(* Logix 5000 project; controller SolisPLC_Vlad_CGL1 vendor 1 type 14 code 226 rev 32.13; software revision 32.02 *)

TASK MainTask (continuous, watchdog 500 ms) : MainProgram, DataLink, Palletizer, Tutorials
TASK SafetyTask (periodic, rate 20 ms, priority 10, watchdog 20 ms, safety) : SafetyProgram

MODULES
   Local : vendor 1 type 14 code 226 (5069 0, rev 32.13)
END_MODULES

TYPE UDT_MQTT_DINT :
STRUCT
   Message : DINT;
   Delay : DINT;
   Timer : TIMER;
   RawData : DINT;
   Delta : DINT;
   OldRawData : DINT;
END_STRUCT
END_TYPE

ADD_ON_INSTRUCTION _AOI_Fah_to_Cel   (* revision 1.0 *)
VAR_INPUT
   Temperature_Fah : REAL; {required}
END_VAR
VAR_OUTPUT
   Temperature_Cel : REAL; {required}
END_VAR
VAR
   Placeholder : REAL; {access None}
   Placeholder1 : REAL; {access None}
END_VAR

ROUTINE Logic   (* ladder *)
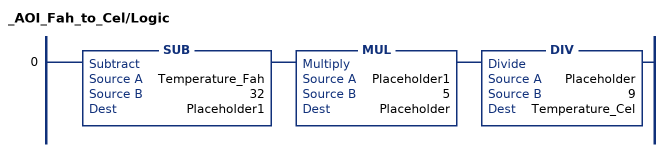
   0: SUB(Temperature_Fah,32,Placeholder1)MUL(Placeholder1,5,Placeholder)DIV(Placeholder,9,Temperature_Cel);
END_ROUTINE
END_ADD_ON_INSTRUCTION

VAR_GLOBAL   (* controller tags *)
   MQTT_OUT : UDT_MQTT_DINT[100] := ([0].Message := 2380, [0].Timer.EN := 1, [0].Timer.TT := 1, [0].RawData := 2380, [0].OldRawData := 2380, [1].Message := 10, [1].Timer.EN := 1, [1].Timer.TT := 1, [1].RawData := 10, [1].OldRawData := 10, [2].Message := 28, [2].Timer.EN := 1, [2].Timer.TT := 1, [2].RawData := 28, [2].OldRawData := 28, [3].Message := 3361, [3].Delay := 1000, [3].Timer.PRE := 1000, [3].Timer.ACC := 633, [3].Timer.EN := 1, [3].Timer.TT := 1, [3].RawData := 3994, [3].Delta := 1000, [3].OldRawData := 3361, [4].Delay := 1000, [4].Timer.PRE := 1000, [4].Timer.ACC := 994, [4].Timer.EN := 1, [4].Timer.TT := 1, [4].Delta := 1000, [5].Timer.EN := 1, [5].Timer.TT := 1, [6].Timer.EN := 1, [6].Timer.TT := 1, [7].Timer.EN := 1, [7].Timer.TT := 1, [8].Timer.EN := 1, [8].Timer.TT := 1, [9].Timer.EN := 1, [9].Timer.TT := 1, [10].Timer.EN := 1, [10].Timer.TT := 1, [11].Timer.EN := 1, [11].Timer.TT := 1, [12].Timer.EN := 1, [12].Timer.TT := 1, [13].Timer.EN := 1, [13].Timer.TT := 1, [14].Timer.EN := 1, [14].Timer.TT := 1, [15].Timer.EN := 1, [15].Timer.TT := 1, [16].Timer.EN := 1, [16].Timer.TT := 1, [17].Timer.EN := 1, [17].Timer.TT := 1, [18].Timer.EN := 1, [18].Timer.TT := 1, [19].Timer.EN := 1, [19].Timer.TT := 1,
        [20].Timer.EN := 1, [20].Timer.TT := 1, [21].Timer.EN := 1, [21].Timer.TT := 1, [22].Timer.EN := 1, [22].Timer.TT := 1, [23].Timer.EN := 1, [23].Timer.TT := 1, [24].Timer.EN := 1, [24].Timer.TT := 1, [25].Timer.EN := 1, [25].Timer.TT := 1, [26].Timer.EN := 1, [26].Timer.TT := 1, [27].Timer.EN := 1, [27].Timer.TT := 1, [28].Timer.EN := 1, [28].Timer.TT := 1, [29].Timer.EN := 1, [29].Timer.TT := 1, [30].Timer.EN := 1, [30].Timer.TT := 1, [31].Timer.EN := 1, [31].Timer.TT := 1, [32].Timer.EN := 1, [32].Timer.TT := 1, [33].Timer.EN := 1, [33].Timer.TT := 1, [34].Timer.EN := 1, [34].Timer.TT := 1, [35].Timer.EN := 1, [35].Timer.TT := 1, [36].Timer.EN := 1, [36].Timer.TT := 1, [37].Timer.EN := 1, [37].Timer.TT := 1, [38].Timer.EN := 1, [38].Timer.TT := 1, [39].Timer.EN := 1, [39].Timer.TT := 1, [40].Timer.EN := 1, [40].Timer.TT := 1, [41].Timer.EN := 1, [41].Timer.TT := 1, [42].Timer.EN := 1, [42].Timer.TT := 1, [43].Timer.EN := 1, [43].Timer.TT := 1, [44].Timer.EN := 1, [44].Timer.TT := 1, [45].Timer.EN := 1, [45].Timer.TT := 1, [46].Timer.EN := 1, [46].Timer.TT := 1, [47].Timer.EN := 1, [47].Timer.TT := 1, [48].Timer.EN := 1, [48].Timer.TT := 1, [49].Timer.EN := 1, [49].Timer.TT := 1,
        [50].Timer.EN := 1, [50].Timer.TT := 1, [51].Timer.EN := 1, [51].Timer.TT := 1, [52].Timer.EN := 1, [52].Timer.TT := 1, [53].Timer.EN := 1, [53].Timer.TT := 1, [54].Timer.EN := 1, [54].Timer.TT := 1, [55].Timer.EN := 1, [55].Timer.TT := 1, [56].Timer.EN := 1, [56].Timer.TT := 1, [57].Timer.EN := 1, [57].Timer.TT := 1, [58].Timer.EN := 1, [58].Timer.TT := 1, [59].Timer.EN := 1, [59].Timer.TT := 1, [60].Timer.EN := 1, [60].Timer.TT := 1, [61].Timer.EN := 1, [61].Timer.TT := 1, [62].Timer.EN := 1, [62].Timer.TT := 1, [63].Timer.EN := 1, [63].Timer.TT := 1, [64].Timer.EN := 1, [64].Timer.TT := 1, [65].Timer.EN := 1, [65].Timer.TT := 1, [66].Timer.EN := 1, [66].Timer.TT := 1, [67].Timer.EN := 1, [67].Timer.TT := 1, [68].Timer.EN := 1, [68].Timer.TT := 1, [69].Timer.EN := 1, [69].Timer.TT := 1, [70].Timer.EN := 1, [70].Timer.TT := 1, [71].Timer.EN := 1, [71].Timer.TT := 1, [72].Timer.EN := 1, [72].Timer.TT := 1, [73].Timer.EN := 1, [73].Timer.TT := 1, [74].Timer.EN := 1, [74].Timer.TT := 1, [75].Timer.EN := 1, [75].Timer.TT := 1, [76].Timer.EN := 1, [76].Timer.TT := 1, [77].Timer.EN := 1, [77].Timer.TT := 1, [78].Timer.EN := 1, [78].Timer.TT := 1, [79].Timer.EN := 1, [79].Timer.TT := 1,
        [80].Timer.EN := 1, [80].Timer.TT := 1, [81].Timer.EN := 1, [81].Timer.TT := 1, [82].Timer.EN := 1, [82].Timer.TT := 1, [83].Timer.EN := 1, [83].Timer.TT := 1, [84].Timer.EN := 1, [84].Timer.TT := 1, [85].Timer.EN := 1, [85].Timer.TT := 1, [86].Timer.EN := 1, [86].Timer.TT := 1, [87].Timer.EN := 1, [87].Timer.TT := 1, [88].Timer.EN := 1, [88].Timer.TT := 1, [89].Timer.EN := 1, [89].Timer.TT := 1, [90].Timer.EN := 1, [90].Timer.TT := 1, [91].Timer.EN := 1, [91].Timer.TT := 1, [92].Timer.EN := 1, [92].Timer.TT := 1, [93].Timer.EN := 1, [93].Timer.TT := 1, [94].Timer.EN := 1, [94].Timer.TT := 1, [95].Timer.EN := 1, [95].Timer.TT := 1, [96].Timer.EN := 1, [96].Timer.TT := 1, [97].Timer.EN := 1, [97].Timer.TT := 1, [98].Timer.EN := 1, [98].Timer.TT := 1, [99].Timer.EN := 1, [99].Timer.TT := 1);
   MQTT_OUT_B : DINT[100];
   MQTT_OUT_BOOL : UDT_MQTT_DINT[100] := ([0].Message := 2252, [0].RawData := 2252);
   MQTT_OUT_DINT : DINT[100] := ([0] := 30869, [1] := 30869, [2] := 10869);
   Pal_D : DINT[100] := ([0] := 2252, [1] := 10, [2] := 28);
        [0].0   // Palletizer Infeed - Start PB
        [0].1   // Palletizer Infeed - Stop PB
        [0].10   // Palletizer Discharge - Stop PB
        [0].11   // Palletizer Discharge - Running Status
        [0].12   // Palletizer Discharge - Full Pallet Ready
        [0].2   // Palletizer Infeed - Enabled Status
        [0].3   // Palletizer Infeed - Full Status
        [0].4   // Palletizer Robot - Start PB
        [0].5   // Palletizer Robot - Stop PB
        [0].6   // Palletizer Robot - Enabled Status
        [0].7   // Palletizer Robot - Pick Up Cases
        [0].8   // Palletizer Robot - Cases On Arm
        [0].9   // Palletizer Discharge - Start PB
   Pal_T : TIMER[100] := ([0].PRE := 1000, [1].PRE := 4268, [1].ACC := 4127, [1].EN := 1, [1].TT := 1, [2].PRE := 6639, [3].PRE := 7587);
   Sys_Timer : TIMER[100] := ([0].PRE := 100000, [0].ACC := 30893, [0].EN := 1, [0].TT := 1, [1].PRE := 500000, [1].ACC := 30893, [1].EN := 1, [1].TT := 1, [2].PRE := 11000, [2].ACC := 10893, [2].EN := 1, [2].TT := 1);
END_VAR

PROGRAM DataLink   (* main routine _01_Main *)
VAR
   index : DINT := 85;
END_VAR

ROUTINE _01_Main   (* ladder *)
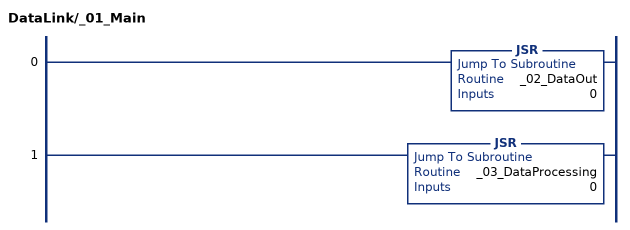
   0: JSR(_02_DataOut,0);
   1: JSR(_03_DataProcessing,0);
END_ROUTINE

ROUTINE _02_DataOut   (* ladder *)
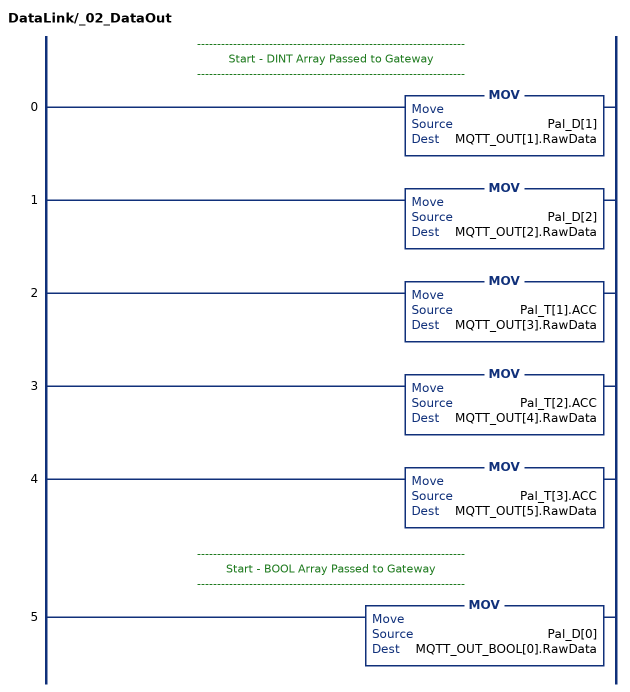
   // -------------------------------------------------------------------
   // Start - DINT Array Passed to Gateway
   // -------------------------------------------------------------------
   0: MOV(Pal_D[1],MQTT_OUT[1].RawData);
   1: MOV(Pal_D[2],MQTT_OUT[2].RawData);
   2: MOV(Pal_T[1].ACC,MQTT_OUT[3].RawData);
   3: MOV(Pal_T[2].ACC,MQTT_OUT[4].RawData);
   4: MOV(Pal_T[3].ACC,MQTT_OUT[5].RawData);
   // -------------------------------------------------------------------
   // Start - BOOL Array Passed to Gateway
   // -------------------------------------------------------------------
   5: MOV(Pal_D[0],MQTT_OUT_BOOL[0].RawData);
END_ROUTINE

ROUTINE _03_DataProcessing   (* ladder *)
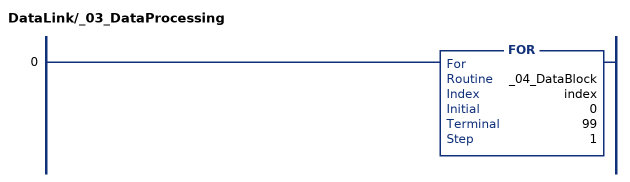
   0: FOR(_04_DataBlock,index,0,99,1);
END_ROUTINE

ROUTINE _04_DataBlock   (* ladder *)
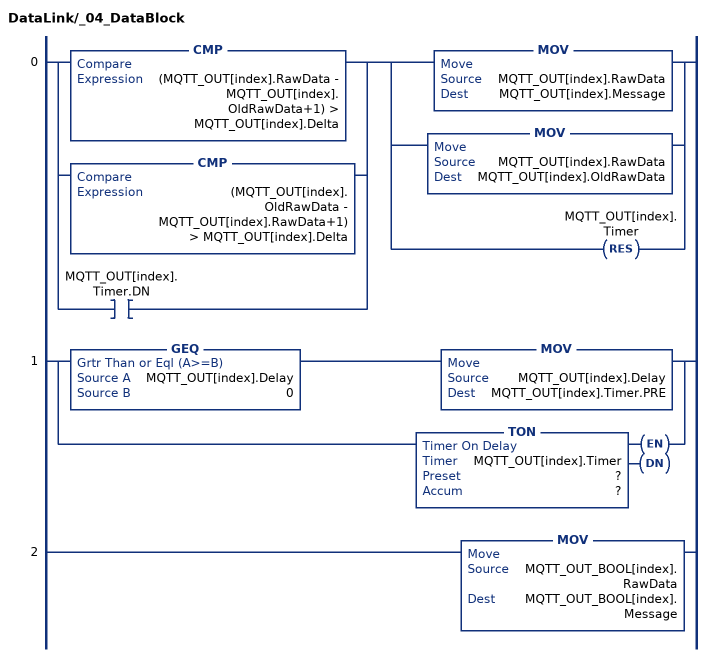
   0: [CMP((MQTT_OUT[index].RawData - MQTT_OUT[index].OldRawData+1) > MQTT_OUT[index].Delta) ,CMP((MQTT_OUT[index].OldRawData - MQTT_OUT[index].RawData+1) > MQTT_OUT[index].Delta) ,XIC(MQTT_OUT[index].Timer.DN) ][MOV(MQTT_OUT[index].RawData,MQTT_OUT[index].Message) ,MOV(MQTT_OUT[index].RawData,MQTT_OUT[index].OldRawData) ,RES(MQTT_OUT[index].Timer) ];
   1: [GEQ(MQTT_OUT[index].Delay,0) MOV(MQTT_OUT[index].Delay,MQTT_OUT[index].Timer.PRE) ,TON(MQTT_OUT[index].Timer,?,?) ];
   2: MOV(MQTT_OUT_BOOL[index].RawData,MQTT_OUT_BOOL[index].Message);
END_ROUTINE
END_PROGRAM

PROGRAM MainProgram   (* main routine MainRoutine *)

ROUTINE MainRoutine   (* ladder *)
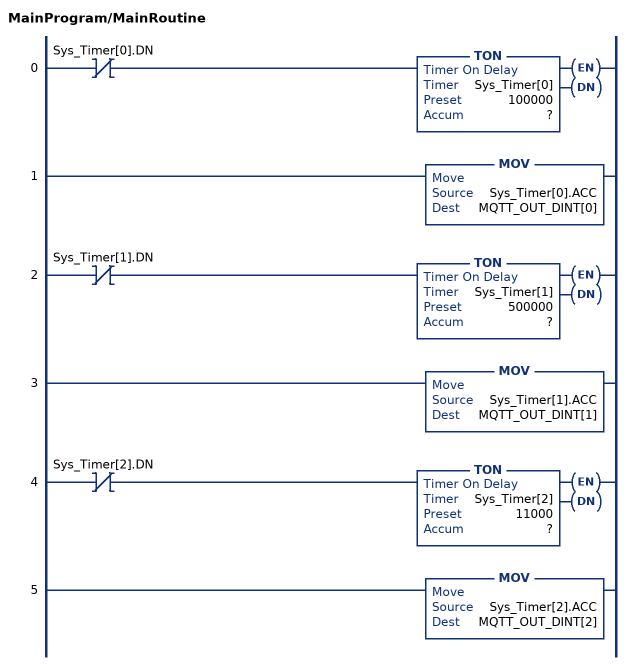
   0: XIO(Sys_Timer[0].DN)TON(Sys_Timer[0],?,?);
   1: MOV(Sys_Timer[0].ACC,MQTT_OUT_DINT[0]);
   2: XIO(Sys_Timer[1].DN)TON(Sys_Timer[1],?,?);
   3: MOV(Sys_Timer[1].ACC,MQTT_OUT_DINT[1]);
   4: XIO(Sys_Timer[2].DN)TON(Sys_Timer[2],?,?);
   5: MOV(Sys_Timer[2].ACC,MQTT_OUT_DINT[2]);
END_ROUTINE
END_PROGRAM

PROGRAM Palletizer   (* main routine _01_Main *)
VAR
   Mask : DINT[20];
   Mask1 : DINT;
   NumberofCasesAtInfeed : DINT := 10;
   Pal_ONS : BOOL[64] := ([0] := 1);
   RandomNum : DINT := 164444007;
   ScanTime : DINT := 204;
   SystemFaulted : BOOL;
   SystemIdle : BOOL;
   SystemRunning : BOOL;
   SystemStatus : DINT;
   Time : DINT[7] := ([0] := 2000, [1] := 1, [2] := 29, [3] := 17, [4] := 51, [5] := 11, [6] := 89702);
END_VAR

ROUTINE _01_Main   (* ladder *)
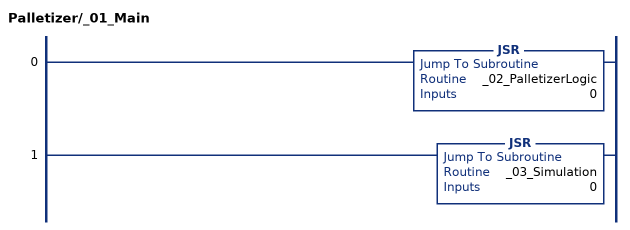
   0: JSR(_02_PalletizerLogic,0);
   1: JSR(_03_Simulation,0);
END_ROUTINE

ROUTINE _02_PalletizerLogic   (* ladder *)
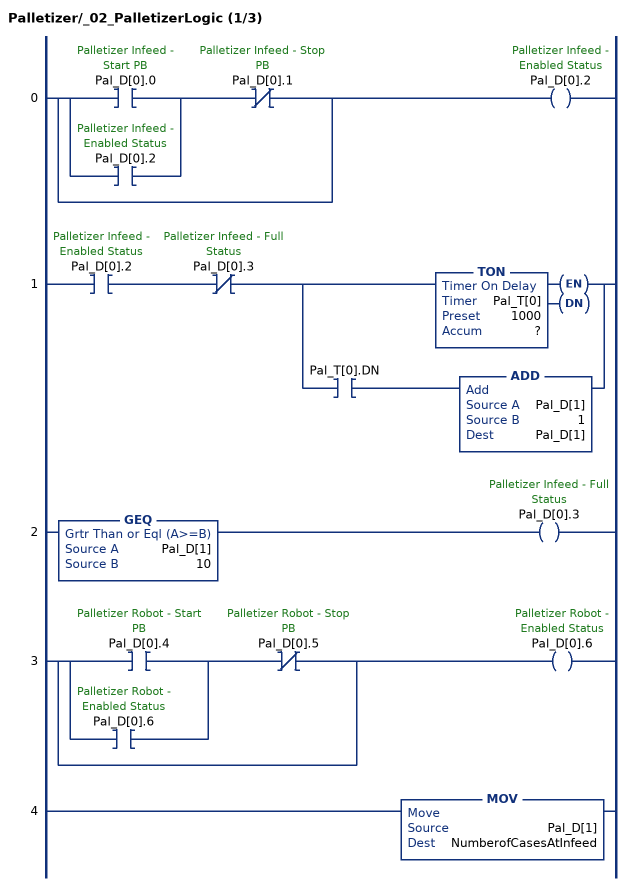
   0: [[XIC(Pal_D[0].0) ,XIC(Pal_D[0].2) ] XIO(Pal_D[0].1) ,]OTE(Pal_D[0].2);
   1: XIC(Pal_D[0].2)XIO(Pal_D[0].3)[TON(Pal_T[0],?,?) ,XIC(Pal_T[0].DN) ADD(Pal_D[1],1,Pal_D[1]) ];
   2: GEQ(Pal_D[1],10)OTE(Pal_D[0].3);
   3: [[XIC(Pal_D[0].4) ,XIC(Pal_D[0].6) ] XIO(Pal_D[0].5) ,]OTE(Pal_D[0].6);
   4: MOV(Pal_D[1],NumberofCasesAtInfeed);
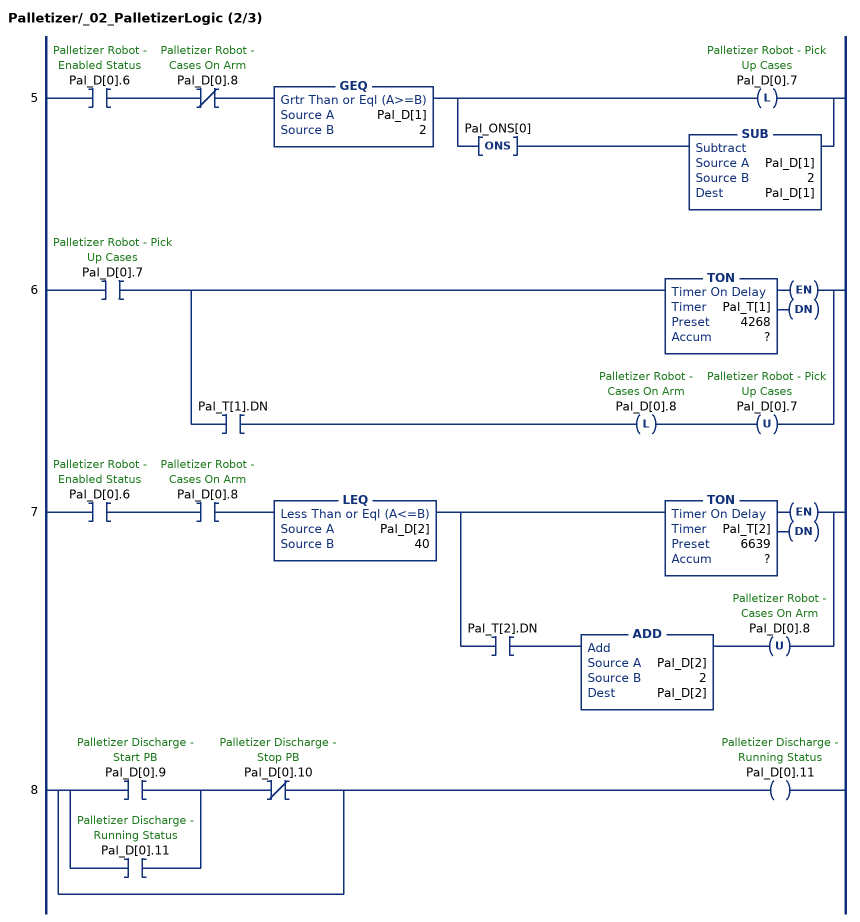
   5: XIC(Pal_D[0].6)XIO(Pal_D[0].8)GEQ(Pal_D[1],2)[OTL(Pal_D[0].7) ,ONS(Pal_ONS[0]) SUB(Pal_D[1],2,Pal_D[1]) ];
   6: XIC(Pal_D[0].7)[TON(Pal_T[1],?,?) ,XIC(Pal_T[1].DN) OTL(Pal_D[0].8) OTU(Pal_D[0].7) ];
   7: XIC(Pal_D[0].6)XIC(Pal_D[0].8)LEQ(Pal_D[2],40)[TON(Pal_T[2],?,?) ,XIC(Pal_T[2].DN) ADD(Pal_D[2],2,Pal_D[2]) OTU(Pal_D[0].8) ];
   8: [[XIC(Pal_D[0].9) ,XIC(Pal_D[0].11) ] XIO(Pal_D[0].10) ,]OTE(Pal_D[0].11);
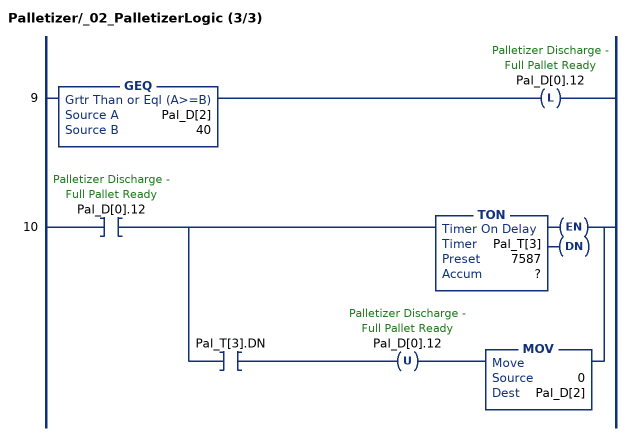
   9: GEQ(Pal_D[2],40)OTL(Pal_D[0].12);
   10: XIC(Pal_D[0].12)[TON(Pal_T[3],?,?) ,XIC(Pal_T[3].DN) OTU(Pal_D[0].12) MOV(0,Pal_D[2]) ];
END_ROUTINE

ROUTINE _03_Simulation   (* ladder *)
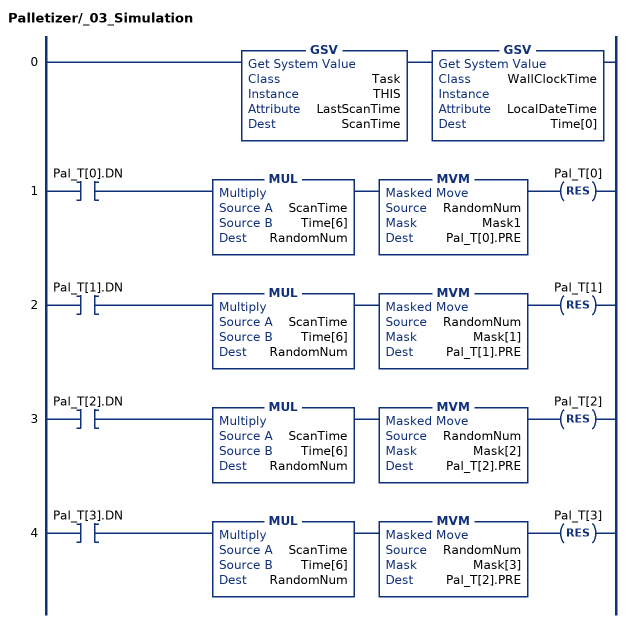
   0: GSV(Task,THIS,LastScanTime,ScanTime)GSV(WallClockTime,,LocalDateTime,Time[0]);
   1: XIC(Pal_T[0].DN)MUL(ScanTime,Time[6],RandomNum)MVM(RandomNum,Mask1,Pal_T[0].PRE)RES(Pal_T[0]);
   2: XIC(Pal_T[1].DN)MUL(ScanTime,Time[6],RandomNum)MVM(RandomNum,Mask[1],Pal_T[1].PRE)RES(Pal_T[1]);
   3: XIC(Pal_T[2].DN)MUL(ScanTime,Time[6],RandomNum)MVM(RandomNum,Mask[2],Pal_T[2].PRE)RES(Pal_T[2]);
   4: XIC(Pal_T[3].DN)MUL(ScanTime,Time[6],RandomNum)MVM(RandomNum,Mask[3],Pal_T[2].PRE)RES(Pal_T[3]);
END_ROUTINE
END_PROGRAM

PROGRAM SafetyProgram   (* main routine MainRoutine, safety *)

ROUTINE MainRoutine   (* ladder *)
END_ROUTINE
END_PROGRAM

PROGRAM Tutorials   (* main routine _01_Main *)
VAR
   _AOI_Fah_to_Cel1 : _AOI_Fah_to_Cel := (Temperature_Fah := 100.0, Temperature_Cel := 37.77778);
   _AOI_Fah_to_Cel2 : _AOI_Fah_to_Cel := (Temperature_Cel := -17.777779);
   Placeholder1 : REAL := -32.0;
   Placeholder2 : REAL := -160.0;
   TempC1 : REAL := -17.777779;
   TempC2 : REAL := 37.77778;
   TempC3 : REAL := -17.777779;
   TempF1 : REAL;
   TempF2 : REAL := 100.0;
   TempF3 : REAL;
END_VAR

ROUTINE _01_Main   (* ladder *)
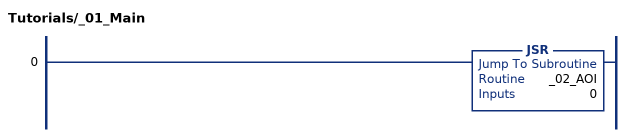
   0: JSR(_02_AOI,0);
END_ROUTINE

ROUTINE _02_AOI   (* ladder *)
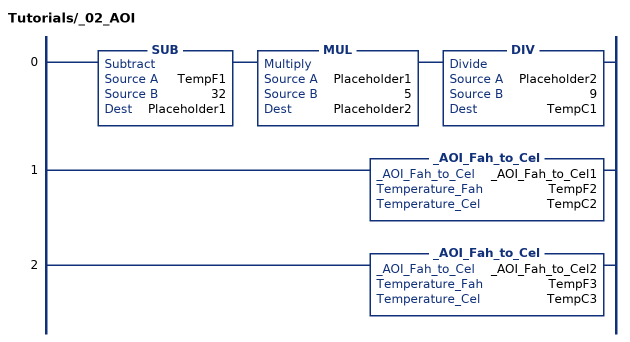
   0: SUB(TempF1,32,Placeholder1)MUL(Placeholder1,5,Placeholder2)DIV(Placeholder2,9,TempC1);
   1: _AOI_Fah_to_Cel(_AOI_Fah_to_Cel1,TempF2,TempC2);
   2: _AOI_Fah_to_Cel(_AOI_Fah_to_Cel2,TempF3,TempC3);
END_ROUTINE
END_PROGRAM
